FUNCTION_BLOCK FB_CylinderBase 
VAR_INPUT
	i_en					:BOOL;
	ref_stCyl              : REFERENCE TO ST_Cylinder;  // 綁定目標 
END_VAR
VAR
    // 既有：除抖與監看 
	_tonTimeOutEnd,_tonEndDeb		:TON;	
	_tonTimeOutORI,_tonORIDeb		:TON;
    // === ConsistencyCheck 專用的「保留狀態」 === 
    _cc_tonStuck   : TON;   // 感測卡住用；放在 FB 內才能跨掃描記憶 
	
	
END_VAR

IF NOT i_en THEN
	RETURN;
END_IF

// === 確認使用的型號 ===  
CASE ref_stCyl.stCylinderPara.eCylinderType OF 
	E_CylinderType.ThreePort_TwoPosition:
		ThreePort_TwoPosition();
	E_CylinderType.FivePort_TwoPosition:
		FivePort_TwoPosition();
END_CASE

_cc_tonStuck(IN:= ref_stCyl.iEndSensor AND ref_stCyl.iOriginSensor , PT:=T#0.3S);
IF _cc_tonStuck.Q THEN
	ref_stCyl.eCylFault	:= E_CylFault.BothSensorsOn;
END_IF
IF ref_stCyl.bReset THEN
	ref_stCyl.bReset:=FALSE;
	Reset();
END_IF


_UpdateFaultFlag();

METHOD PRIVATE _UpdateFaultFlag : BOOL
VAR_INPUT
END_VAR
ref_stCyl.bError := (ref_stCyl.eCylFault <> E_CylFault.None) ;
END_METHOD

METHOD INTERNAL FivePort_TwoPosition
VAR_INPUT
END_VAR
//異常感測時間	
	_tonTimeOutEnd(IN := ref_stCyl.qExtendCoil AND NOT ref_stCyl.iEndSensor, PT := ref_stCyl.stCylinderPara.tEndTimeout);
	
	IF _tonTimeOutEnd.Q AND NOT ref_stCyl.stCylinderPara.bEndNoSensor THEN		//確認TimeOut + NO Sensor 
		ref_stCyl.eCylFault := E_CylFault.TimeoutExtend;
	END_IF

	_tonTimeOutORI(IN := ref_stCyl.qRetractCoil AND NOT ref_stCyl.iOriginSensor, PT := ref_stCyl.stCylinderPara.tOriginTimeout);
	
	IF _tonTimeOutORI.Q AND NOT ref_stCyl.stCylinderPara.bOriginNoSensor THEN		//確認TimeOut + NO Sensor 
		ref_stCyl.eCylFault := E_CylFault.TimeoutRetract;
	END_IF	

	
//穩定時間 輸出監控 
	
	IF NOT ref_stCyl.stCylinderPara.bEndNoSensor  THEN			//有感測器 
		_tonEndDeb(IN:=ref_stCyl.iEndSensor , PT := ref_stCyl.stCylinderPara.tEndDebounceTime );
		ref_stCyl.bEndConfirmed	:= _tonEndDeb.Q ;
	ELSE														//沒感測器 
		_tonEndDeb(IN:=ref_stCyl.qExtendCoil , PT := ref_stCyl.stCylinderPara.tEndDebounceTime );
		ref_stCyl.bEndConfirmed	:= _tonEndDeb.Q ;		
	END_IF

	
//穩定時間 回歸

	IF NOT ref_stCyl.stCylinderPara.bOriginNoSensor  THEN			//有感測器 
		_tonORIDeb(IN:=ref_stCyl.iOriginSensor , PT := ref_stCyl.stCylinderPara.tOriginDebounceTime );
		ref_stCyl.bOriginConfirmed	:= _tonORIDeb.Q ;
	ELSE														//沒感測器  
		_tonORIDeb(IN:= ref_stCyl.qRetractCoil , PT := ref_stCyl.stCylinderPara.tOriginDebounceTime );
		ref_stCyl.bOriginConfirmed	:= _tonORIDeb.Q ;		
	END_IF
//自動關閉 
	IF ref_stCyl.stCylinderPara.bCoilAutoOff THEN
		IF ref_stCyl.iEndSensor	THEN
			ref_stCyl.qExtendCoil :=FALSE;
		END_IF
		IF ref_stCyl.iOriginSensor	THEN
			ref_stCyl.qRetractCoil :=FALSE;
		END_IF	
	
	END_IF
END_METHOD

METHOD Home : BOOL
VAR_INPUT
END_VAR
CASE ref_stCyl.stCylinderPara.eCylinderType OF 
	E_CylinderType.ThreePort_TwoPosition:
		ref_stCyl.qExtendCoil	:=FALSE;
	E_CylinderType.FivePort_TwoPosition:
		ref_stCyl.qExtendCoil	:=FALSE;
		ref_stCyl.qRetractCoil	:= TRUE;
END_CASE
Home:= ref_stCyl.iOriginSensor;
END_METHOD

METHOD Reset
VAR_INPUT
END_VAR
// ======================================================
//  Reset  — 復歸：清錯 + 停止所有監看/定時器
// ======================================================
(*
// 停止監看
_watchOri := FALSE;
_watchEnd := FALSE;

// 關閉所有 TON
_tonTO_Ori(IN := FALSE);
_tonTO_End(IN := FALSE);
_tonOriDeb(IN := FALSE);
_tonEndDeb(IN := FALSE);
_cc_tonStuck(IN := FALSE);

*)
// 清除錯誤/故障碼
ref_stCyl.eCylFault      := E_CylFault.None;
ref_stCyl.bError         := FALSE;

// （可選）清除已確認狀態，讓到位需重新經過除抖
ref_stCyl.bOriginConfirmed := FALSE;
ref_stCyl.bEndConfirmed    := FALSE;
END_METHOD

METHOD INTERNAL ThreePort_TwoPosition
VAR_INPUT
END_VAR
//異常感測時間	
	_tonTimeOutEnd(IN := ref_stCyl.qExtendCoil AND NOT ref_stCyl.iEndSensor, PT := ref_stCyl.stCylinderPara.tEndTimeout);
	
	IF _tonTimeOutEnd.Q AND NOT ref_stCyl.stCylinderPara.bEndNoSensor THEN		//確認TimeOut + NO Sensor 
		ref_stCyl.eCylFault := E_CylFault.TimeoutExtend;
	END_IF

	_tonTimeOutORI(IN := NOT ref_stCyl.qExtendCoil AND NOT ref_stCyl.iOriginSensor, PT := ref_stCyl.stCylinderPara.tOriginTimeout);
	
	IF _tonTimeOutORI.Q AND NOT ref_stCyl.stCylinderPara.bOriginNoSensor THEN		//確認TimeOut + NO Sensor 
		ref_stCyl.eCylFault := E_CylFault.TimeoutRetract;
	END_IF	

	
//穩定時間 輸出監控 
	
	IF NOT ref_stCyl.stCylinderPara.bEndNoSensor  THEN			//有感測器 
		_tonEndDeb(IN:=ref_stCyl.iEndSensor , PT := ref_stCyl.stCylinderPara.tEndDebounceTime );
		ref_stCyl.bEndConfirmed	:= _tonEndDeb.Q ;
	ELSE														//沒感測器 
		_tonEndDeb(IN:=ref_stCyl.qExtendCoil , PT := ref_stCyl.stCylinderPara.tEndDebounceTime );
		ref_stCyl.bEndConfirmed	:= _tonEndDeb.Q ;		
	END_IF

	
//穩定時間 回歸

	IF NOT ref_stCyl.stCylinderPara.bOriginNoSensor  THEN			//有感測器 
		_tonORIDeb(IN:=ref_stCyl.iOriginSensor , PT := ref_stCyl.stCylinderPara.tOriginDebounceTime );
		ref_stCyl.bOriginConfirmed	:= _tonORIDeb.Q ;
	ELSE														//沒感測器  
		_tonORIDeb(IN:=NOT ref_stCyl.qExtendCoil , PT := ref_stCyl.stCylinderPara.tOriginDebounceTime );
		ref_stCyl.bOriginConfirmed	:= _tonORIDeb.Q ;		
	END_IF
END_METHOD

END_FUNCTION_BLOCK

(* stored: Version 1.1.0.1, ProductVersion 3.1.4024.15
   POU FB_CylinderBase: Id {97fb96fe-ea69-4de0-bfa5-ae51e7218c65}, SpecialFunc None
   Method _UpdateFaultFlag: Id {4b601817-3cd7-4932-862b-12560673e7f2}
   Method FivePort_TwoPosition: Id {804f7a54-f6f1-4ac6-84c8-f91a3881ee6e}
   Method Home: Id {12ecb7da-4fa2-4989-bf54-16ddc6ce5cc4}
   Method Reset: Id {a023ba7c-23c1-4fb5-8466-5cfa667519a2}
   Method ThreePort_TwoPosition: Id {b4ab4507-2acc-4b60-a06b-0fa2c5650d46} *)
